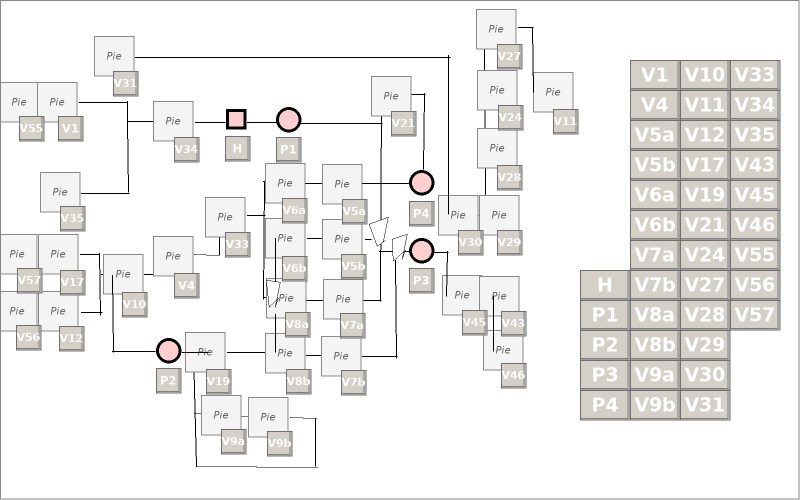
VISUALIZATION Screen_3_Sub_1  // 800x500
    Line (411,94) (425,94)
    Line (424,93) (423,169)
    Line (380,96) (394,96)
    Line (135,57) (450,57)
    Line (307,238) (342,238)
    Line (42,101) (59,101)
    Line (79,102) (127,102)
    Line (127,121) (175,121)
    Line (81,193) (129,193)
    Line (127,121) (128,192)
    Line (195,122) (225,122)
    Line (247,122) (277,122)
    Line (301,123) (382,123)
    Line (381,96) (380,301)
    Line (380,183) (410,183)
    Line (379,251) (409,251)
    Line (363,300) (381,300)
    Line (306,300) (347,300)
    Line (304,183) (345,183)
    Line (264,181) (263,299)
    Line (263,181) (288,181)
    Line (263,297) (288,297)
    Line (306,355) (341,355)
    Line (275,238) (290,238)
    Line (362,356) (397,356)
    Line (38,254) (59,254)
    Line (39,311) (60,311)
    Line (80,254) (99,254)
    Line (81,312) (102,312)
    Line (101,274) (123,274)
    Line (160,256) (174,255)
    Line (144,274) (162,274)
    Line (160,256) (160,275)
    Line (217,217) (226,217)
    Line (194,254) (218,255)
    Line (219,217) (219,255)
    Line (247,215) (265,215)
    Line (112,351) (155,351)
    Line (227,352) (287,352)
    Line (447,213) (460,214)
    Line (477,215) (503,214)
    Line (484,27) (485,215)
    Line (483,148) (498,148)
    Line (483,89) (498,89)
    Line (483,28) (498,28)
    Line (533,91) (555,91)
    Line (483,295) (501,296)
    Line (433,252) (448,252)
    Line (445,295) (465,295)
    Line (492,350) (505,350)
    Line (193,351) (196,466)
    Line (194,413) (224,414)
    Line (241,416) (271,417)
    Line (290,417) (316,418)
    Line (196,466) (317,467)
    Line (365,239) (371,239)
    Pie (-1,82 40x40), colour toggle: GVL.HMI_Maintenance_V55
    Pie (37,82 40x40), colour toggle: GVL.HMI_Maintenance_V1
    Pie (94,36 40x40), colour toggle: GVL.HMI_Maintenance_V31
    Pie (153,101 40x40), colour toggle: GVL.HMI_Maintenance_V34
    Pie (40,172 40x40), colour toggle: GVL.HMI_Maintenance_V35
    Pie (-3,234 40x40), colour toggle: GVL.HMI_Maintenance_V57
    Pie (-3,291 40x40), colour toggle: GVL.HMI_Maintenance_V56
    Pie (38,234 40x40), colour toggle: GVL.HMI_Maintenance_V17
    Pie (38,291 40x40), colour toggle: GVL.HMI_Maintenance_V12
    Pie (371,76 40x40), colour toggle: GVL.HMI_Maintenance_V21
    Pie (476,9 40x40), colour toggle: GVL.HMI_Maintenance_V27
    Pie (477,70 40x40), colour toggle: GVL.HMI_Maintenance_V24
    Pie (477,128 40x40), colour toggle: GVL.HMI_Maintenance_V28
    Pie (533,72 40x40), colour toggle: GVL.HMI_Maintenance_V11
    Button (580,270 50x30), "H", colour toggle: GVL.HMI_Maintenance_H
        toggle GVL.HMI_Maintenance_H p2164770859=TRUE
    Button (580,300 50x30), "P1", colour toggle: GVL.HMI_Maintenance_P1
        toggle GVL.HMI_Maintenance_P1 p2164770859=TRUE
    Button (580,330 50x30), "P2", colour toggle: GVL.HMI_Maintenance_P2
        toggle GVL.HMI_Maintenance_P2 p2164770859=TRUE
    Button (580,360 50x30), "P3", colour toggle: GVL.HMI_Maintenance_P3
        toggle GVL.HMI_Maintenance_P3 p2164770859=TRUE
    Button (580,390 50x30), "P4", colour toggle: GVL.HMI_Maintenance_P4
        toggle GVL.HMI_Maintenance_P4 p2164770859=TRUE
    Button (630,270 50x30), "V7b", colour toggle: GVL.HMI_Maintenance_V7B
        toggle GVL.HMI_Maintenance_V7B p2164770859=TRUE
    Button (630,300 50x30), "V8a", colour toggle: GVL.HMI_Maintenance_V8A
        toggle GVL.HMI_Maintenance_V8A p2164770859=TRUE
    Button (630,330 50x30), "V8b", colour toggle: GVL.HMI_Maintenance_V8B
        toggle GVL.HMI_Maintenance_V8B p2164770859=TRUE
    Button (630,360 50x30), "V9a", colour toggle: GVL.HMI_Maintenance_V9A
        toggle GVL.HMI_Maintenance_V9A p2164770859=TRUE
    Button (630,390 50x30), "V9b", colour toggle: GVL.HMI_Maintenance_V9B
        toggle GVL.HMI_Maintenance_V9B p2164770859=TRUE
    Button (630,120 50x30), "V5a", colour toggle: GVL.HMI_Maintenance_V5A
        toggle GVL.HMI_Maintenance_V5A p2164770859=TRUE
    Button (630,150 50x30), "V5b", colour toggle: GVL.HMI_Maintenance_V5B
        toggle GVL.HMI_Maintenance_V5B p2164770859=TRUE
    Button (630,180 50x30), "V6a", colour toggle: GVL.HMI_Maintenance_V6A
        toggle GVL.HMI_Maintenance_V6A p2164770859=TRUE
    Button (630,210 50x30), "V6b", colour toggle: GVL.HMI_Maintenance_V6B
        toggle GVL.HMI_Maintenance_V6B p2164770859=TRUE
    Button (630,240 50x30), "V7a", colour toggle: GVL.HMI_Maintenance_V7A
        toggle GVL.HMI_Maintenance_V7A p2164770859=TRUE
    Button (630,60 50x30), "V1", colour toggle: GVL.HMI_Maintenance_V1
        toggle GVL.HMI_Maintenance_V1 p2164770859=TRUE
    Button (630,90 50x30), "V4", colour toggle: GVL.HMI_Maintenance_V4
        toggle GVL.HMI_Maintenance_V4 p2164770859=TRUE
    Button (680,270 50x30), "V27", colour toggle: GVL.HMI_Maintenance_V27
        toggle GVL.HMI_Maintenance_V27 p2164770859=TRUE
    Button (680,300 50x30), "V28", colour toggle: GVL.HMI_Maintenance_V28
        toggle GVL.HMI_Maintenance_V28 p2164770859=TRUE
    Button (680,330 50x30), "V29", colour toggle: GVL.HMI_Maintenance_V29
        toggle GVL.HMI_Maintenance_V29 p2164770859=TRUE
    Button (680,360 50x30), "V30", colour toggle: GVL.HMI_Maintenance_V30
        toggle GVL.HMI_Maintenance_V30 p2164770859=TRUE
    Button (680,390 50x30), "V31", colour toggle: GVL.HMI_Maintenance_V31
        toggle GVL.HMI_Maintenance_V31 p2164770859=TRUE
    Button (680,120 50x30), "V12", colour toggle: GVL.HMI_Maintenance_V12
        toggle GVL.HMI_Maintenance_V12 p2164770859=TRUE
    Button (680,150 50x30), "V17", colour toggle: GVL.HMI_Maintenance_V17
        toggle GVL.HMI_Maintenance_V17 p2164770859=TRUE
    Button (680,180 50x30), "V19", colour toggle: GVL.HMI_Maintenance_V19
        toggle GVL.HMI_Maintenance_V19 p2164770859=TRUE
    Button (680,210 50x30), "V21", colour toggle: GVL.HMI_Maintenance_V21
        toggle GVL.HMI_Maintenance_V21 p2164770859=TRUE
    Button (680,240 50x30), "V24", colour toggle: GVL.HMI_Maintenance_V24
        toggle GVL.HMI_Maintenance_V24 p2164770859=TRUE
    Button (680,60 50x30), "V10", colour toggle: GVL.HMI_Maintenance_V10
        toggle GVL.HMI_Maintenance_V10 p2164770859=TRUE
    Button (680,90 50x30), "V11", colour toggle: GVL.HMI_Maintenance_V11
        toggle GVL.HMI_Maintenance_V11 p2164770859=TRUE
    Button (730,270 50x30), "V56", colour toggle: GVL.HMI_Maintenance_V56
        toggle GVL.HMI_Maintenance_V56 p2164770859=TRUE
    Button (730,300 50x30), "V57", colour toggle: GVL.HMI_Maintenance_V57
        toggle GVL.HMI_Maintenance_V57 p2164770859=TRUE
    Button (730,120 50x30), "V35", colour toggle: GVL.HMI_Maintenance_V35
        toggle GVL.HMI_Maintenance_V35 p2164770859=TRUE
    Button (730,150 50x30), "V43", colour toggle: GVL.HMI_Maintenance_V43
        toggle GVL.HMI_Maintenance_V43 p2164770859=TRUE
    Button (730,180 50x30), "V45", colour toggle: GVL.HMI_Maintenance_V45
        toggle GVL.HMI_Maintenance_V45 p2164770859=TRUE
    Button (730,210 50x30), "V46", colour toggle: GVL.HMI_Maintenance_V46
        toggle GVL.HMI_Maintenance_V46 p2164770859=TRUE
    Button (730,240 50x30), "V55", colour toggle: GVL.HMI_Maintenance_V55
        toggle GVL.HMI_Maintenance_V55 p2164770859=TRUE
    Button (730,60 50x30), "V33", colour toggle: GVL.HMI_Maintenance_V33
        toggle GVL.HMI_Maintenance_V33 p2164770859=TRUE
    Button (730,90 50x30), "V34", colour toggle: GVL.HMI_Maintenance_V34
        toggle GVL.HMI_Maintenance_V34 p2164770859=TRUE
    Button (19,116 25x25), "V55", colour toggle: GVL.HMI_Maintenance_V55
        toggle GVL.HMI_Maintenance_V55 p2164770859=TRUE
    Button (58,116 25x25), "V1", colour toggle: GVL.HMI_Maintenance_V1
        toggle GVL.HMI_Maintenance_V1 p2164770859=TRUE
    Button (113,71 25x25), "V31", colour toggle: GVL.HMI_Maintenance_V31
        toggle GVL.HMI_Maintenance_V31 p2164770859=TRUE
    Button (391,111 25x25), "V21", colour toggle: GVL.HMI_Maintenance_V21
        toggle GVL.HMI_Maintenance_V21 p2164770859=TRUE
    Button (497,44 25x25), "V27", colour toggle: GVL.HMI_Maintenance_V27
        toggle GVL.HMI_Maintenance_V27 p2164770859=TRUE
    Button (498,105 25x25), "V24", colour toggle: GVL.HMI_Maintenance_V24
        toggle GVL.HMI_Maintenance_V24 p2164770859=TRUE
    Button (497,165 25x25), "V28", colour toggle: GVL.HMI_Maintenance_V28
        toggle GVL.HMI_Maintenance_V28 p2164770859=TRUE
    Button (553,109 25x25), "V11", colour toggle: GVL.HMI_Maintenance_V11
        toggle GVL.HMI_Maintenance_V11 p2164770859=TRUE
    Button (174,137 25x25), "V34", colour toggle: GVL.HMI_Maintenance_V34
        toggle GVL.HMI_Maintenance_V34 p2164770859=TRUE
    Button (60,206 25x25), "V35", colour toggle: GVL.HMI_Maintenance_V35
        toggle GVL.HMI_Maintenance_V35 p2164770859=TRUE
    Button (17,268 25x25), "V57", colour toggle: GVL.HMI_Maintenance_V57
        toggle GVL.HMI_Maintenance_V57 p2164770859=TRUE
    Button (60,270 25x25), "V17", colour toggle: GVL.HMI_Maintenance_V17
        toggle GVL.HMI_Maintenance_V17 p2164770859=TRUE
    Button (16,325 25x25), "V56", colour toggle: GVL.HMI_Maintenance_V56
        toggle GVL.HMI_Maintenance_V56 p2164770859=TRUE
    Button (59,326 25x25), "V12", colour toggle: GVL.HMI_Maintenance_V12
        toggle GVL.HMI_Maintenance_V12 p2164770859=TRUE
    Rectangle (226,109 20x20), colour toggle: GVL.HMI_Maintenance_H
    Button (225,136 25x25), "H", colour toggle: GVL.HMI_Maintenance_H
        toggle GVL.HMI_Maintenance_H p2164770859=TRUE
    Ellipse (276,107 25x25), colour toggle: GVL.HMI_Maintenance_P1
    Button (276,137 25x25), "P1", colour toggle: GVL.HMI_Maintenance_P1
        toggle GVL.HMI_Maintenance_P1 p2164770859=TRUE
    Ellipse (156,338 25x25), colour toggle: GVL.HMI_Maintenance_P2
    Button (156,368 25x25), "P2", colour toggle: GVL.HMI_Maintenance_P2
        toggle GVL.HMI_Maintenance_P2 p2164770859=TRUE
    Ellipse (409,238 25x25), colour toggle: GVL.HMI_Maintenance_P3
    Ellipse (409,170 25x25), colour toggle: GVL.HMI_Maintenance_P4
    Button (409,201 25x25), "P4", colour toggle: GVL.HMI_Maintenance_P4
        toggle GVL.HMI_Maintenance_P4 p2164770859=TRUE
    Button (409,268 25x25), "P3", colour toggle: GVL.HMI_Maintenance_P3
        toggle GVL.HMI_Maintenance_P3 p2164770859=TRUE
    Pie (153,236 40x40), colour toggle: GVL.HMI_Maintenance_V4
    Button (174,273 25x25), "V4", colour toggle: GVL.HMI_Maintenance_V4
        toggle GVL.HMI_Maintenance_V4 p2164770859=TRUE
    Pie (103,254 40x40), colour toggle: GVL.HMI_Maintenance_V10
    Button (122,292 25x25), "V10", colour toggle: GVL.HMI_Maintenance_V10
        toggle GVL.HMI_Maintenance_V10 p2164770859=TRUE
    Pie (185,332 40x40), colour toggle: GVL.HMI_Maintenance_V19
    Button (206,369 25x25), "V19", colour toggle: GVL.HMI_Maintenance_V19
        toggle GVL.HMI_Maintenance_V19 p2164770859=TRUE
    Pie (479,195 40x40), colour toggle: GVL.HMI_Maintenance_V29
    Button (497,230 25x25), "V29", colour toggle: GVL.HMI_Maintenance_V29
        toggle GVL.HMI_Maintenance_V29 p2164770859=TRUE
    Pie (438,195 40x40), colour toggle: GVL.HMI_Maintenance_V30
    Button (458,230 25x25), "V30", colour toggle: GVL.HMI_Maintenance_V30
        toggle GVL.HMI_Maintenance_V30 p2164770859=TRUE
    Pie (205,197 40x40), colour toggle: GVL.HMI_Maintenance_V33
    Button (225,232 25x25), "V33", colour toggle: GVL.HMI_Maintenance_V33
        toggle GVL.HMI_Maintenance_V33 p2164770859=TRUE
    Pie (442,275 40x40), colour toggle: GVL.HMI_Maintenance_V45
    Pie (479,276 40x40), colour toggle: GVL.HMI_Maintenance_V43
    Pie (483,330 40x40), colour toggle: GVL.HMI_Maintenance_V46
    Button (462,310 25x25), "V45", colour toggle: GVL.HMI_Maintenance_V45
        toggle GVL.HMI_Maintenance_V45 p2164770859=TRUE
    Button (501,311 25x25), "V43", colour toggle: GVL.HMI_Maintenance_V43
        toggle GVL.HMI_Maintenance_V43 p2164770859=TRUE
    Button (501,363 25x25), "V46", colour toggle: GVL.HMI_Maintenance_V46
        toggle GVL.HMI_Maintenance_V46 p2164770859=TRUE
    Pie (265,163 40x40), colour toggle: GVL.HMI_Maintenance_V6A
    Pie (322,164 40x40), colour toggle: GVL.HMI_Maintenance_V5A
    Pie (265,218 40x40), colour toggle: GVL.HMI_Maintenance_V6B
    Pie (322,219 40x40), colour toggle: GVL.HMI_Maintenance_V5B
    Pie (266,278 40x40), colour toggle: GVL.HMI_Maintenance_V8A
    Pie (323,279 40x40), colour toggle: GVL.HMI_Maintenance_V7A
    Pie (265,333 40x40), colour toggle: GVL.HMI_Maintenance_V8B
    Pie (321,336 40x40), colour toggle: GVL.HMI_Maintenance_V7B
    Button (342,199 25x25), "V5a", colour toggle: GVL.HMI_Maintenance_V5A
        toggle GVL.HMI_Maintenance_V5A p2164770859=TRUE
    Button (341,254 25x25), "V5b", colour toggle: GVL.HMI_Maintenance_V5B
        toggle GVL.HMI_Maintenance_V5B p2164770859=TRUE
    Button (282,198 25x25), "V6a", colour toggle: GVL.HMI_Maintenance_V6A
        toggle GVL.HMI_Maintenance_V6A p2164770859=TRUE
    Button (282,256 25x25), "V6b", colour toggle: GVL.HMI_Maintenance_V6B
        toggle GVL.HMI_Maintenance_V6B p2164770859=TRUE
    Button (340,313 25x25), "V7a", colour toggle: GVL.HMI_Maintenance_V7A
        toggle GVL.HMI_Maintenance_V7A p2164770859=TRUE
    Button (341,370 25x25), "V7b", colour toggle: GVL.HMI_Maintenance_V7B
        toggle GVL.HMI_Maintenance_V7B p2164770859=TRUE
    Button (285,312 25x25), "V8a", colour toggle: GVL.HMI_Maintenance_V8A
        toggle GVL.HMI_Maintenance_V8A p2164770859=TRUE
    Button (286,369 25x25), "V8b", colour toggle: GVL.HMI_Maintenance_V8B
        toggle GVL.HMI_Maintenance_V8B p2164770859=TRUE
    Pie (201,395 40x40), colour toggle: GVL.HMI_Maintenance_V9A
    Pie (248,397 40x40), colour toggle: GVL.HMI_Maintenance_V9B
    Button (221,429 25x25), "V9a", colour toggle: GVL.HMI_Maintenance_V9A
        toggle GVL.HMI_Maintenance_V9A p2164770859=TRUE
    Button (267,431 25x25), "V9b", colour toggle: GVL.HMI_Maintenance_V9B
        toggle GVL.HMI_Maintenance_V9B p2164770859=TRUE
    Line (127,101) (127,121)
    Line (362,183) (384,183)
    Polygon (392,239) (407,234) (402,259) (405,250) (393,261)
    Line (395,260) (396,358)
    Polygon (369,224) (388,217) (383,242) (385,240) (377,246)
    Line (275,238) (275,290)
    Polygon (266,280) (280,282) (275,307) (278,298) (269,307)
    Line (275,314) (275,352)
    Line (99,253) (100,315)
    Line (112,275) (113,352)
    Line (182,352) (208,352)
    Line (448,55) (448,214)
    Line (518,27) (533,27)
    Line (532,27) (533,92)
    Line (447,251) (446,296)
    Line (493,296) (493,351)
    Line (315,418) (315,466)
END_VISUALIZATION

(* stored: Version 1.1.0.1, ProductVersion 3.1.4024.12
   Visu Screen_3_Sub_1: Id {a76cbaf9-32aa-4394-82ce-a38de2020efe} *)
